FUNCTION_BLOCK ABSTRACT EncodedDrive EXTENDS Drive
VAR_OUTPUT
	position : LREAL;
	targetPos : LREAL;
END_VAR

METHOD ABSTRACT moveAbsolute : BOOL
VAR_INPUT
END_VAR
END_METHOD

END_FUNCTION_BLOCK

(* stored: Version 1.1.0.1, ProductVersion 3.1.4024.11
   POU EncodedDrive: Id {caa7332e-f27e-4d9e-a2f6-47f54869698f}, SpecialFunc None
   Method moveAbsolute: Id {83083c7a-48ec-46dd-9173-7415bee385a6} *)
